// TIA Portal V19 export
TYPE "PositioningMachine_Config"
// stored: Access Published
   STRUCT
      SLS_VEL : LReal;
      DelayMissingCondition : Time := T#3s;   // Delay before rise up missing condition warnings
      Ax : Struct
         OptionON_EncoderSelection : Bool := FALSE;
         OptionON_ParameterChange : Bool := FALSE;
         OptionON_AutoReloadPosition : Bool := FALSE;
         OptionON_ManPreset : Bool := FALSE;
         HomeMode : Int := 0;
         PosAxis : "TAx_Config";
      END_STRUCT;
      Fan : Struct
         Presence : Bool := FALSE;
         DelayOff : Time := T#10M;
      END_STRUCT;
      Brake_Presence : Bool;
   END_STRUCT;
END_TYPE
